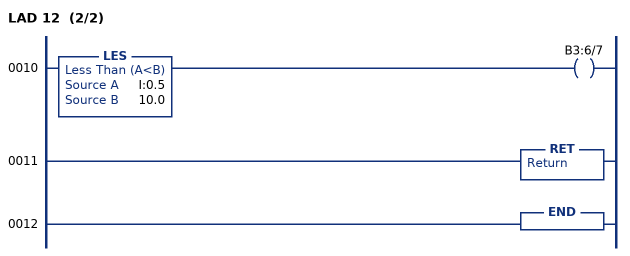
% Rung: 10 %
SOR LES I:0.5 10.0 OTE B3:6/7 EOR
% Rung: 11 %
SOR RET EOR
% Rung: 12 %
SOR END EOR

LADDER 13
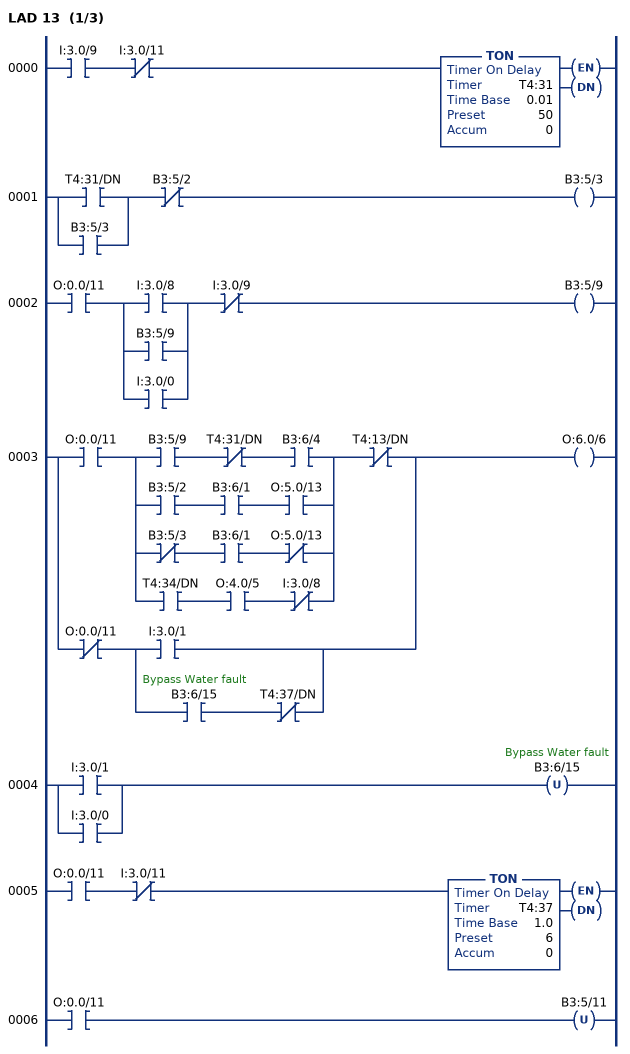
% Rung: 0 %
SOR XIC I:3.0/9 XIO I:3.0/11 TON T4:31 0.01 50 0 EOR
% Rung: 1 %
SOR BST XIC T4:31/DN NXB XIC B3:5/3 BND XIO B3:5/2 OTE B3:5/3 EOR
% Rung: 2 %
SOR XIC O:0.0/11 BST XIC I:3.0/8 NXB BST XIC B3:5/9 NXB XIC I:3.0/0 BND BND XIO I:3.0/9 OTE B3:5/9 EOR
% Rung: 3 %
SOR BST XIC O:0.0/11 BST XIC B3:5/9 XIO T4:31/DN XIC B3:6/4 NXB XIC B3:5/2 XIC B3:6/1 XIC O:5.0/13 NXB BST XIO B3:5/3 XIC B3:6/1 XIO O:5.0/13 NXB XIC T4:34/DN XIC O:4.0/5 XIO I:3.0/8 BND BND XIO T4:13/DN NXB XIO O:0.0/11 BST XIC I:3.0/1 NXB XIC B3:6/15 XIO T4:37/DN BND BND OTE O:6.0/6 EOR
%   B3:6/15  "Bypass Water fault" %
% Rung: 4 %
SOR BST XIC I:3.0/1 NXB XIC I:3.0/0 BND OTU B3:6/15 EOR
%   B3:6/15  "Bypass Water fault" %
% Rung: 5 %
SOR XIC O:0.0/11 XIO I:3.0/11 TON T4:37 1.0 6 0 EOR
% Rung: 6 %
SOR XIC O:0.0/11 OTU B3:5/11 EOR

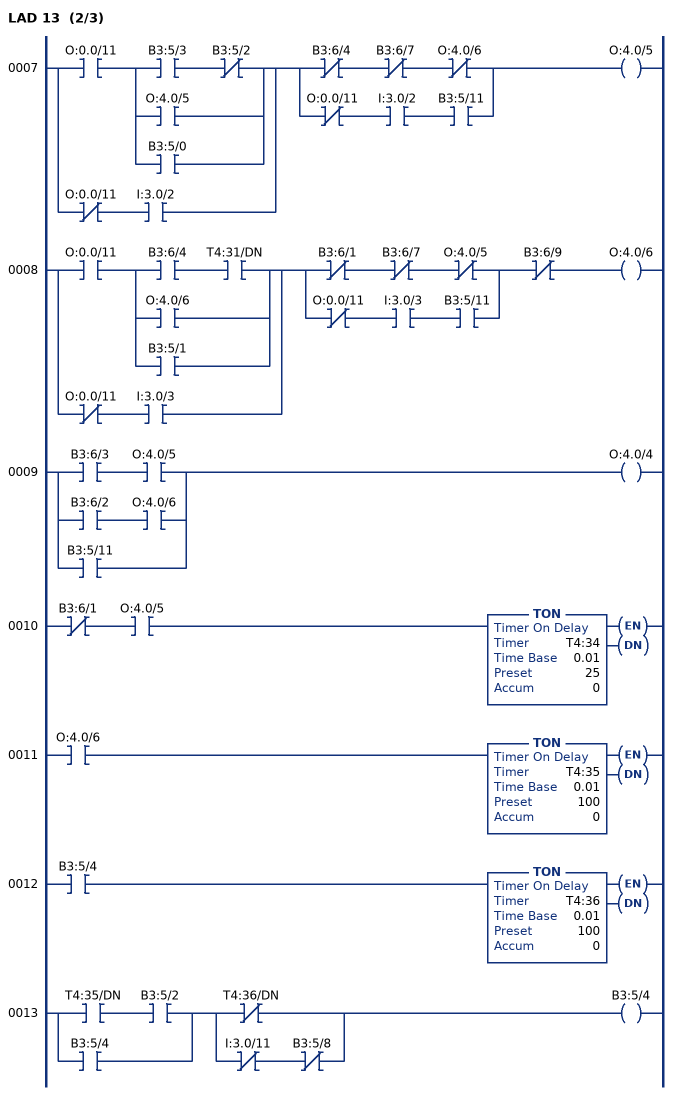
% Rung: 7 %
SOR BST XIC O:0.0/11 BST XIC B3:5/3 XIO B3:5/2 NXB XIC O:4.0/5 NXB XIC B3:5/0 BND NXB XIO O:0.0/11 XIC I:3.0/2 BND BST XIO B3:6/4 XIO B3:6/7 XIO O:4.0/6 NXB XIO O:0.0/11 XIC I:3.0/2 XIC B3:5/11 BND OTE O:4.0/5 EOR
% Rung: 8 %
SOR BST XIC O:0.0/11 BST XIC B3:6/4 XIC T4:31/DN NXB XIC O:4.0/6 NXB XIC B3:5/1 BND NXB XIO O:0.0/11 XIC I:3.0/3 BND BST XIO B3:6/1 XIO B3:6/7 XIO O:4.0/5 NXB XIO O:0.0/11 XIC I:3.0/3 XIC B3:5/11 BND XIO B3:6/9 OTE O:4.0/6 EOR
% Rung: 9 %
SOR BST BST XIC B3:6/3 XIC O:4.0/5 NXB XIC B3:6/2 XIC O:4.0/6 BND NXB XIC B3:5/11 BND OTE O:4.0/4 EOR
% Rung: 10 %
SOR XIO B3:6/1 XIC O:4.0/5 TON T4:34 0.01 25 0 EOR
% Rung: 11 %
SOR XIC O:4.0/6 TON T4:35 0.01 100 0 EOR
% Rung: 12 %
SOR XIC B3:5/4 TON T4:36 0.01 100 0 EOR
% Rung: 13 %
SOR BST XIC T4:35/DN XIC B3:5/2 NXB XIC B3:5/4 BND BST XIO T4:36/DN NXB XIO I:3.0/11 XIO B3:5/8 BND OTE B3:5/4 EOR

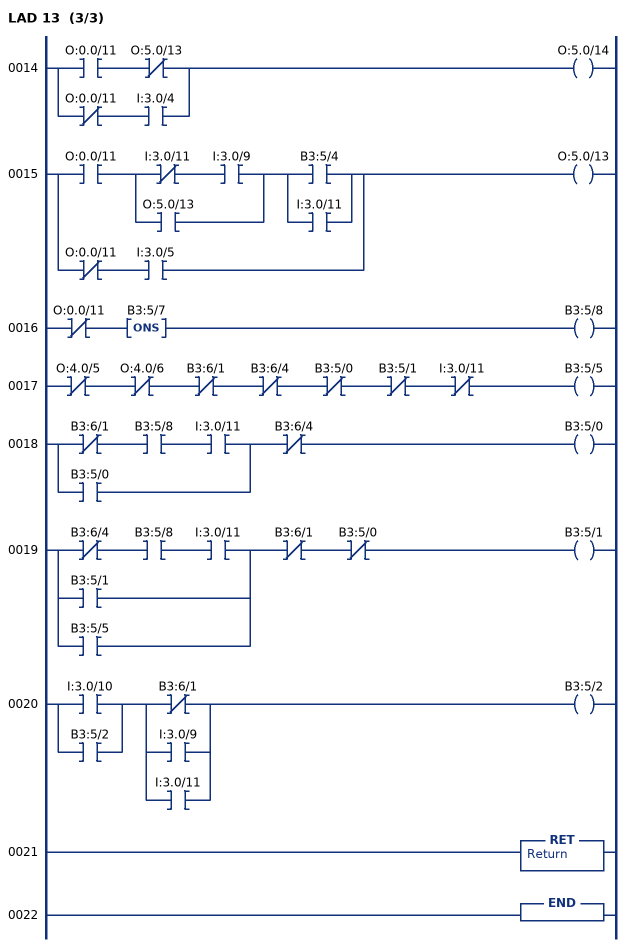
% Rung: 14 %
SOR BST XIC O:0.0/11 XIO O:5.0/13 NXB XIO O:0.0/11 XIC I:3.0/4 BND OTE O:5.0/14 EOR
% Rung: 15 %
SOR BST XIC O:0.0/11 BST XIO I:3.0/11 XIC I:3.0/9 NXB XIC O:5.0/13 BND BST XIC B3:5/4 NXB XIC I:3.0/11 BND NXB XIO O:0.0/11 XIC I:3.0/5 BND OTE O:5.0/13 EOR
% Rung: 16 %
SOR XIO O:0.0/11 ONS B3:5/7 OTE B3:5/8 EOR
% Rung: 17 %
SOR XIO O:4.0/5 XIO O:4.0/6 XIO B3:6/1 XIO B3:6/4 XIO B3:5/0 XIO B3:5/1 XIO I:3.0/11 OTE B3:5/5 EOR
% Rung: 18 %
SOR BST XIO B3:6/1 XIC B3:5/8 XIC I:3.0/11 NXB XIC B3:5/0 BND XIO B3:6/4 OTE B3:5/0 EOR
% Rung: 19 %
SOR BST XIO B3:6/4 XIC B3:5/8 XIC I:3.0/11 NXB XIC B3:5/1 NXB XIC B3:5/5 BND XIO B3:6/1 XIO B3:5/0 OTE B3:5/1 EOR
% Rung: 20 %
SOR BST XIC I:3.0/10 NXB XIC B3:5/2 BND BST XIO B3:6/1 NXB BST XIC I:3.0/9 NXB XIC I:3.0/11 BND BND OTE B3:5/2 EOR
% Rung: 21 %
SOR RET EOR
% Rung: 22 %
SOR END EOR

DATA TABLE (non-zero values as saved)
DATA B3
% B3:0 % 0X5D0A 0X41C3 0X36B8 0X0400 0X0011 0X0082 0X0018
DATA T4
% .PRE .ACC %
% T4:0 % 50 50
% T4:1 % 1 0
% T4:2 % 1 0
% T4:3 % 500 0
% T4:4 % 2 2
% T4:5 % 3 3
% T4:6 % 658 0
% T4:7 % 375 500
% T4:8 % 6 0
% T4:9 % 2 0
% T4:10 % 500 0
% T4:11 % 75 73
% T4:12 % 150 0
% T4:13 % 180 0
% T4:14 % 120 0
% T4:15 % 400 0
% T4:16 % 400 0
% T4:17 % 100 100
% T4:18 % 100 0
% T4:20 % 7 0
% T4:21 % 700 0
% T4:22 % 300 0
% T4:23 % 69 0
% T4:24 % 69 0
% T4:25 % 6 0
% T4:26 % 70 0
% T4:27 % 75 0
% T4:28 % 400 0
% T4:30 % 50 100
% T4:31 % 50 0
% T4:32 % 1 0
% T4:33 % 1 0
% T4:34 % 25 0
% T4:35 % 100 0
% T4:36 % 100 0
% T4:37 % 6 0
DATA N7
% N7:0 % 86 17 10 65 130 21 24 0 69 0
% N7:10 % 9 9 0 0 0 0 0 0 0 0
DATA F8
% F8:0 % 12114 0 0 0 0
% F8:5 % 4071 115.61 35.21321 0 0
% F8:20 % 0.125 0.62 7.25 7.87 7.25
% F8:25 % 27.85 35.1 0 0 35.5
